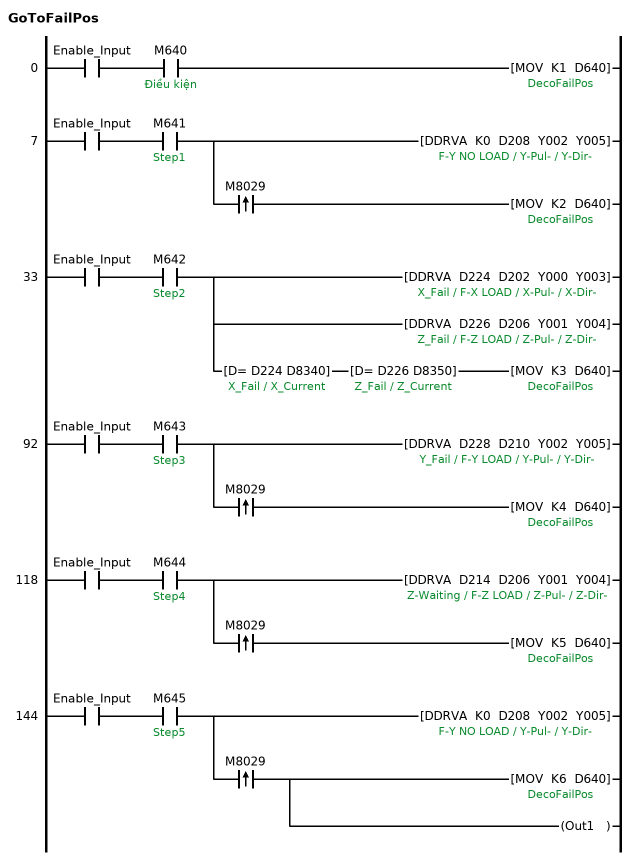
[picture p24: ladder of GoToFailPos, rungs at steps 0 to 144]
0     LD      Enable_Input
      AND     M640  ; Điều kiện
      MOV     K1 D640  ; DecoFailPos
7     LD      Enable_Input
      AND     M641  ; Step1
      DDRVA   K0 D208 Y002 Y005  ; F-Y NO LOAD / Y-Pul- / Y-Dir-
      ANDP    M8029
      MOV     K2 D640
33    LD      Enable_Input
      AND     M642  ; Step2
      DDRVA   D224 D202 Y000 Y003  ; X_Fail / F-X LOAD / X-Pul- / X-Dir-
      DDRVA   D226 D206 Y001 Y004  ; Z_Fail / F-Z LOAD / Z-Pul- / Z-Dir-
      ANDD=   D224 D8340  ; X_Fail / X_Current
      ANDD=   D226 D8350  ; Z_Fail / Z_Current
      MOV     K3 D640
92    LD      Enable_Input
      AND     M643  ; Step3
      DDRVA   D228 D210 Y002 Y005  ; Y_Fail / F-Y LOAD
      ANDP    M8029
      MOV     K4 D640
118   LD      Enable_Input
      AND     M644  ; Step4
      DDRVA   D214 D206 Y001 Y004  ; Z-Waiting
      ANDP    M8029
      MOV     K5 D640
144   LD      Enable_Input
      AND     M645  ; Step5
      DDRVA   K0 D208 Y002 Y005
      ANDP    M8029
      MOV     K6 D640
      OUT     Out1
END_FUNCTION_BLOCK

PROGRAM RETRI
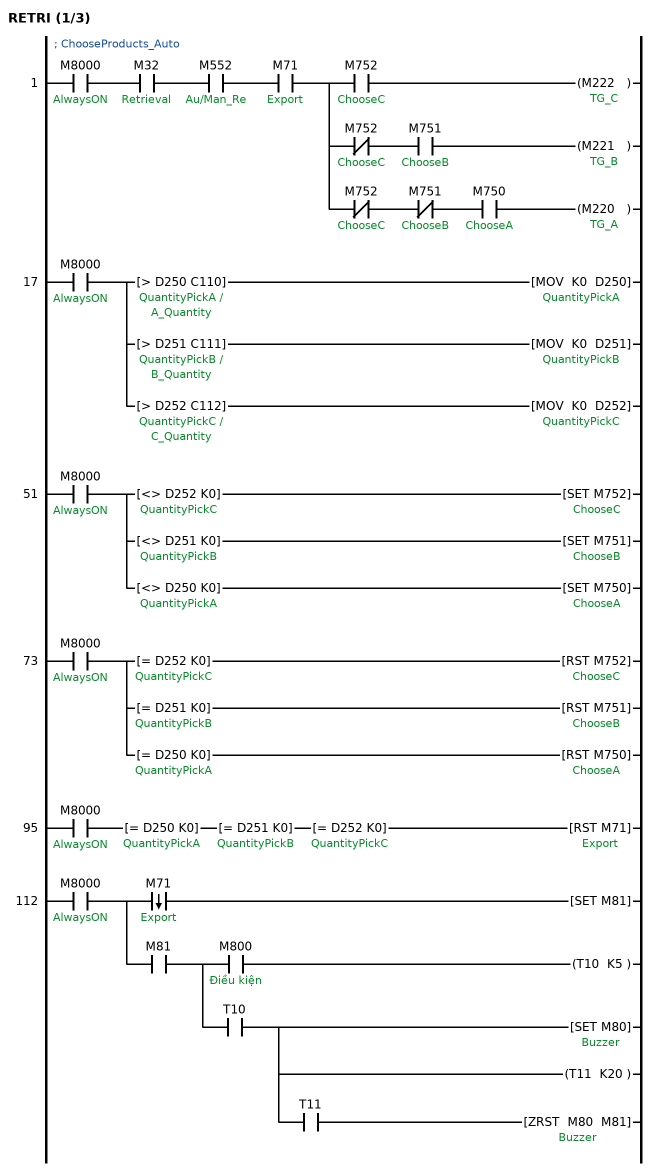
; ChooseProducts_Auto
1     LD      M8000  ; AlwaysON
      AND     M32  ; Retrieval
      AND     M552  ; Au/Man_Re
      AND     M71  ; Export
      MPS
      AND     M752  ; ChooseC
      OUT     M222  ; TG_C
      MRD
      ANI     M752  ; ChooseC
      AND     M751  ; ChooseB
      OUT     M221  ; TG_B
      MPP
      ANI     M752  ; ChooseC
      ANI     M751  ; ChooseB
      AND     M750  ; ChooseA
      OUT     M220  ; TG_A
17    LD      M8000  ; AlwaysON
      MPS
      AND>    D250 C110  ; QuantityPickA / A_Quantity
      MOV     K0 D250
      MRD
      AND>    D251 C111  ; QuantityPickB / B_Quantity
      MOV     K0 D251
      MPP
      AND>    D252 C112  ; QuantityPickC / C_Quantity
      MOV     K0 D252
51    LD      M8000  ; AlwaysON
      MPS
      AND<>   D252 K0  ; QuantityPickC
      SET     M752  ; ChooseC
      MRD
      AND<>   D251 K0  ; QuantityPickB
      SET     M751  ; ChooseB
      MPP
      AND<>   D250 K0  ; QuantityPickA
      SET     M750  ; ChooseA
73    LD      M8000  ; AlwaysON
      MPS
      AND=    D252 K0  ; QuantityPickC
      RST     M752  ; ChooseC
      MRD
      AND=    D251 K0  ; QuantityPickB
      RST     M751  ; ChooseB
      MPP
      AND=    D250 K0  ; QuantityPickA
      RST     M750  ; ChooseA
95    LD      M8000  ; AlwaysON
      AND=    D250 K0  ; QuantityPickA
      AND=    D251 K0  ; QuantityPickB
      AND=    D252 K0  ; QuantityPickC
      RST     M71  ; Export
112   LD      M8000  ; AlwaysON
      MPS
      ANDF    M71  ; Export
      SET     M81
      MPP
      AND     M81
      MPS
      AND     M800  ; Điều kiện
      OUT     T10 K5
      MPP
      AND     T10
      SET     M80  ; Buzzer
      OUT     T11 K20
      AND     T11
      ZRST    M80 M81
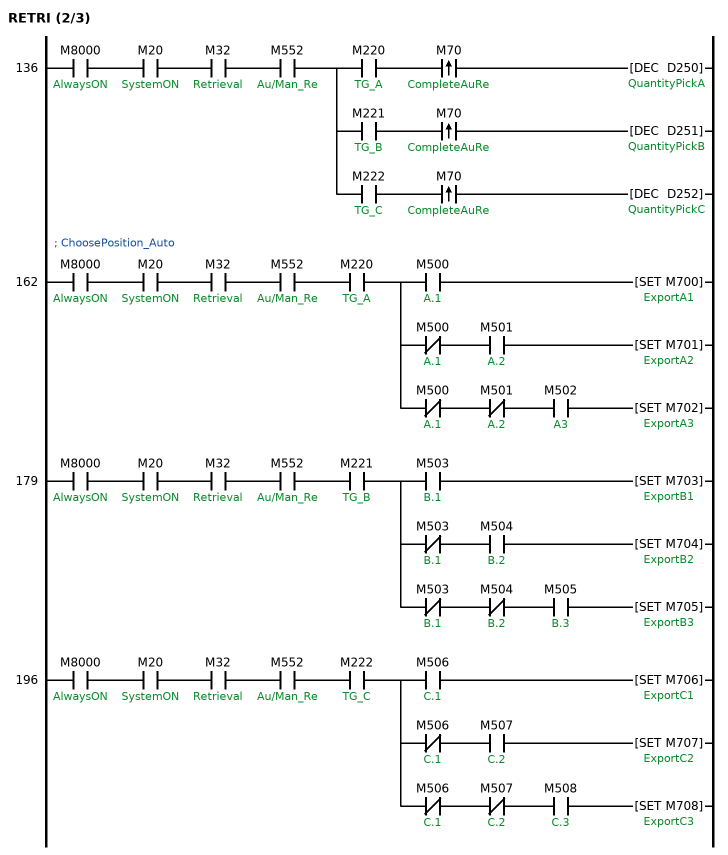
136   LD      M8000  ; AlwaysON
      AND     M20  ; SystemON
      AND     M32  ; Retrieval
      AND     M552  ; Au/Man_Re
      MPS
      AND     M220  ; TG_A
      ANDP    M70  ; CompleteAuRe
      DEC     D250
      MRD
      AND     M221  ; TG_B
      ANDP    M70  ; CompleteAuRe
      DEC     D251
      MPP
      AND     M222  ; TG_C
      ANDP    M70  ; CompleteAuRe
      DEC     D252
; ChoosePosition_Auto
162   LD      M8000  ; AlwaysON
      AND     M20  ; SystemON
      AND     M32  ; Retrieval
      AND     M552  ; Au/Man_Re
      AND     M220  ; TG_A
      MPS
      AND     M500  ; A.1
      SET     M700  ; ExportA1
      MRD
      ANI     M500  ; A.1
      AND     M501  ; A.2
      SET     M701  ; ExportA2
      MPP
      ANI     M500  ; A.1
      ANI     M501  ; A.2
      AND     M502  ; A3
      SET     M702  ; ExportA3
179   LD      M8000  ; AlwaysON
      AND     M20  ; SystemON
      AND     M32  ; Retrieval
      AND     M552  ; Au/Man_Re
      AND     M221  ; TG_B
      MPS
      AND     M503  ; B.1
      SET     M703  ; ExportB1
      MRD
      ANI     M503  ; B.1
      AND     M504  ; B.2
      SET     M704  ; ExportB2
      MPP
      ANI     M503  ; B.1
      ANI     M504  ; B.2
      AND     M505  ; B.3
      SET     M705  ; ExportB3
196   LD      M8000  ; AlwaysON
      AND     M20  ; SystemON
      AND     M32  ; Retrieval
      AND     M552  ; Au/Man_Re
      AND     M222  ; TG_C
      MPS
      AND     M506  ; C.1
      SET     M706  ; ExportC1
      MRD
      ANI     M506  ; C.1
      AND     M507  ; C.2
      SET     M707  ; ExportC2
      MPP
      ANI     M506  ; C.1
      ANI     M507  ; C.2
      AND     M508  ; C.3
      SET     M708  ; ExportC3
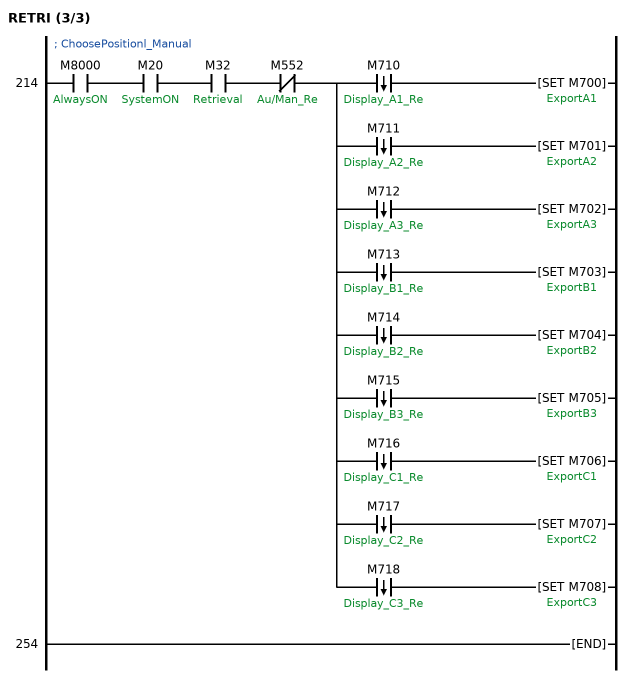
; ChoosePositionl_Manual
214   LD      M8000  ; AlwaysON
      AND     M20  ; SystemON
      AND     M32  ; Retrieval
      ANI     M552  ; Au/Man_Re
      MPS
      ANDF    M710  ; Display_A1_Re
      SET     M700  ; ExportA1
      MRD
      ANDF    M711  ; Display_A2_Re
      SET     M701  ; ExportA2
      MRD
      ANDF    M712  ; Display_A3_Re
      SET     M702  ; ExportA3
      MRD
      ANDF    M713  ; Display_B1_Re
      SET     M703  ; ExportB1
      MRD
      ANDF    M714  ; Display_B2_Re
      SET     M704  ; ExportB2
      MRD
      ANDF    M715  ; Display_B3_Re
      SET     M705  ; ExportB3
      MRD
      ANDF    M716  ; Display_C1_Re
      SET     M706  ; ExportC1
      MRD
      ANDF    M717  ; Display_C2_Re
      SET     M707  ; ExportC2
      MPP
      ANDF    M718  ; Display_C3_Re
      SET     M708  ; ExportC3
254   END
END_PROGRAM

PROGRAM Display
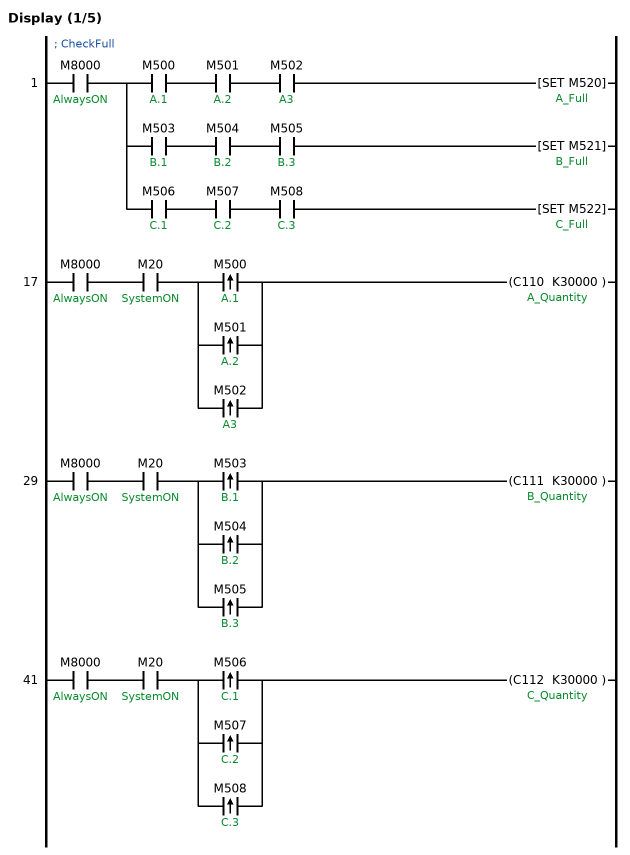
; CheckFull
1     LD      M8000  ; AlwaysON
      MPS
      AND     M500  ; A.1
      AND     M501  ; A.2
      AND     M502  ; A3
      SET     M520  ; A_Full
      MRD
      AND     M503  ; B.1
      AND     M504  ; B.2
      AND     M505  ; B.3
      SET     M521  ; B_Full
      MPP
      AND     M506  ; C.1
      AND     M507  ; C.2
      AND     M508  ; C.3
      SET     M522  ; C_Full
17    LD      M8000  ; AlwaysON
      AND     M20  ; SystemON
      LDP     M500  ; A.1
      ORP     M501  ; A.2
      ORP     M502  ; A3
      ANB
      OUT     C110 K30000  ; A_Quantity
29    LD      M8000  ; AlwaysON
      AND     M20  ; SystemON
      LDP     M503  ; B.1
      ORP     M504  ; B.2
      ORP     M505  ; B.3
      ANB
      OUT     C111 K30000  ; B_Quantity
41    LD      M8000  ; AlwaysON
      AND     M20  ; SystemON
      LDP     M506  ; C.1
      ORP     M507  ; C.2
      ORP     M508  ; C.3
      ANB
      OUT     C112 K30000  ; C_Quantity
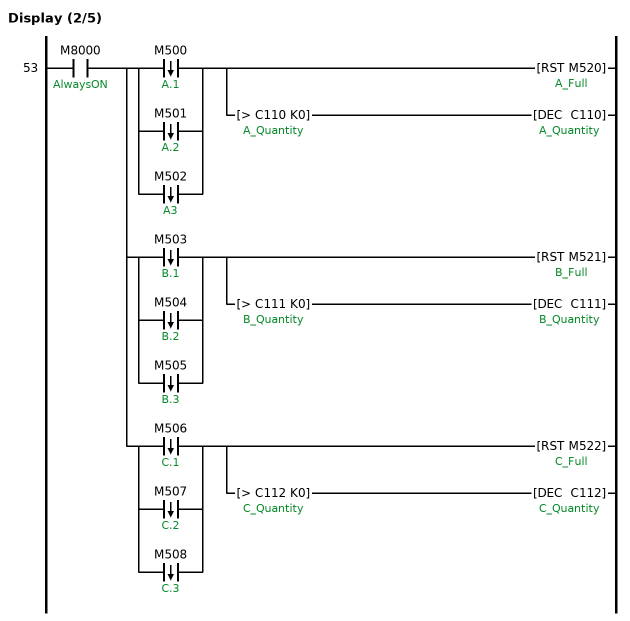
53    LD      M8000  ; AlwaysON
      MPS
      LDF     M500  ; A.1
      ORF     M501  ; A.2
      ORF     M502  ; A3
      ANB
      RST     M520  ; A_Full
      AND>    C110 K0  ; A_Quantity
      DEC     C110
      MRD
      LDF     M503  ; B.1
      ORF     M504  ; B.2
      ORF     M505  ; B.3
      ANB
      RST     M521  ; B_Full
      AND>    C111 K0  ; B_Quantity
      DEC     C111
      MPP
      LDF     M506  ; C.1
      ORF     M507  ; C.2
      ORF     M508  ; C.3
      ANB
      RST     M522  ; C_Full
      AND>    C112 K0  ; C_Quantity
      DEC     C112
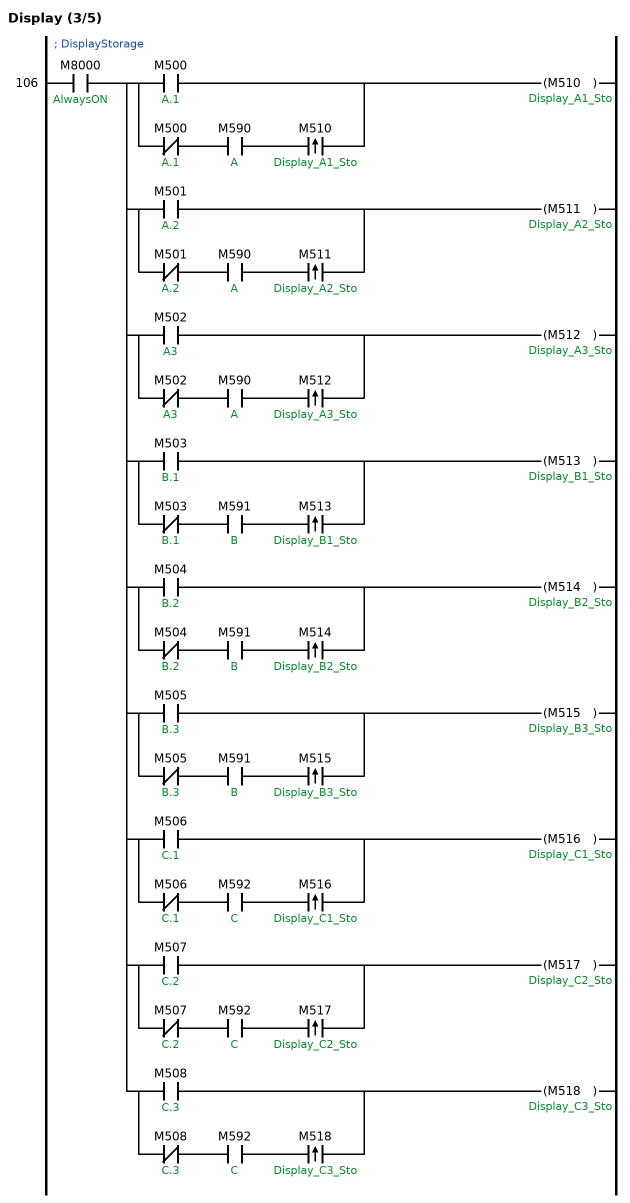
; DisplayStorage
106   LD      M8000  ; AlwaysON
      MPS
      LD      M500  ; A.1
      LDI     M500  ; A.1
      AND     M590  ; A
      ANDP    M510  ; Display_A1_Sto
      ORB
      ANB
      OUT     M510  ; Display_A1_Sto
      MRD
      LD      M501  ; A.2
      LDI     M501  ; A.2
      AND     M590  ; A
      ANDP    M511  ; Display_A2_Sto
      ORB
      ANB
      OUT     M511  ; Display_A2_Sto
      MRD
      LD      M502  ; A3
      LDI     M502  ; A3
      AND     M590  ; A
      ANDP    M512  ; Display_A3_Sto
      ORB
      ANB
      OUT     M512  ; Display_A3_Sto
      MRD
      LD      M503  ; B.1
      LDI     M503  ; B.1
      AND     M591  ; B
      ANDP    M513  ; Display_B1_Sto
      ORB
      ANB
      OUT     M513  ; Display_B1_Sto
      MRD
      LD      M504  ; B.2
      LDI     M504  ; B.2
      AND     M591  ; B
      ANDP    M514  ; Display_B2_Sto
      ORB
      ANB
      OUT     M514  ; Display_B2_Sto
      MRD
      LD      M505  ; B.3
      LDI     M505  ; B.3
      AND     M591  ; B
      ANDP    M515  ; Display_B3_Sto
      ORB
      ANB
      OUT     M515  ; Display_B3_Sto
      MRD
      LD      M506  ; C.1
      LDI     M506  ; C.1
      AND     M592  ; C
      ANDP    M516  ; Display_C1_Sto
      ORB
      ANB
      OUT     M516  ; Display_C1_Sto
      MRD
      LD      M507  ; C.2
      LDI     M507  ; C.2
      AND     M592  ; C
      ANDP    M517  ; Display_C2_Sto
      ORB
      ANB
      OUT     M517  ; Display_C2_Sto
      MPP
      LD      M508  ; C.3
      LDI     M508  ; C.3
      AND     M592  ; C
      ANDP    M518  ; Display_C3_Sto
      ORB
      ANB
      OUT     M518  ; Display_C3_Sto
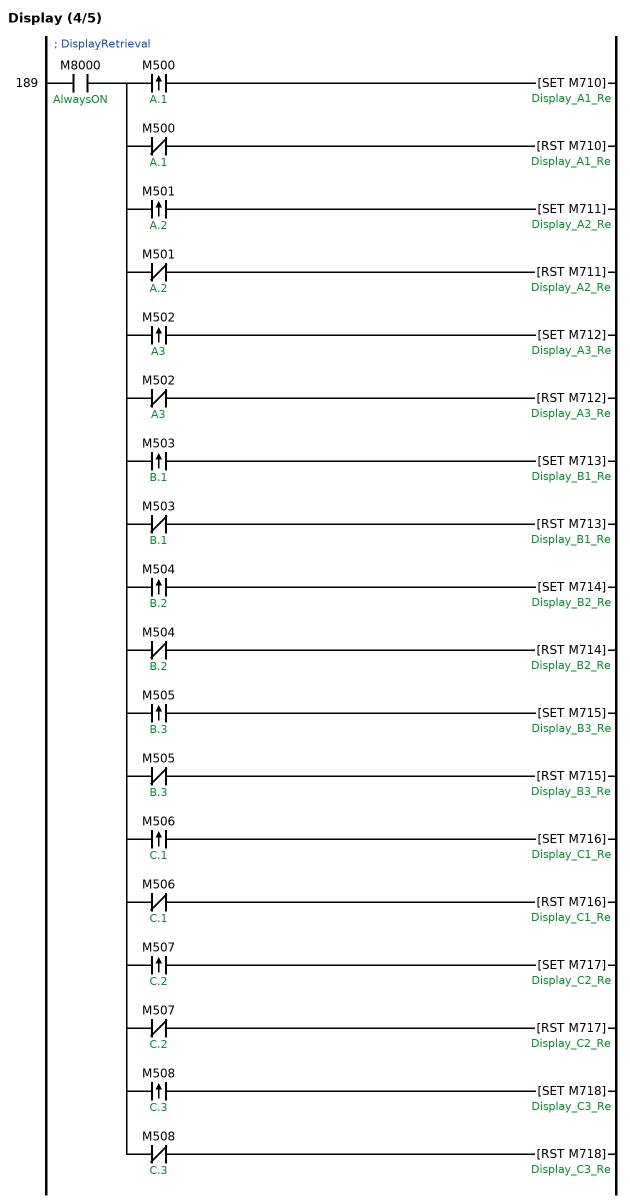
; DisplayRetrieval
189   LD      M8000  ; AlwaysON
      MPS
      ANDP    M500  ; A.1
      SET     M710  ; Display_A1_Re
      MRD
      ANI     M500  ; A.1
      RST     M710  ; Display_A1_Re
      MRD
      ANDP    M501  ; A.2
      SET     M711  ; Display_A2_Re
      MRD
      ANI     M501  ; A.2
      RST     M711  ; Display_A2_Re
      MRD
      ANDP    M502  ; A3
      SET     M712  ; Display_A3_Re
      MRD
      ANI     M502  ; A3
      RST     M712  ; Display_A3_Re
      MRD
      ANDP    M503  ; B.1
      SET     M713  ; Display_B1_Re
      MRD
      ANI     M503  ; B.1
      RST     M713  ; Display_B1_Re
      MRD
      ANDP    M504  ; B.2
      SET     M714  ; Display_B2_Re
      MRD
      ANI     M504  ; B.2
      RST     M714  ; Display_B2_Re
      MRD
      ANDP    M505  ; B.3
      SET     M715  ; Display_B3_Re
      MRD
      ANI     M505  ; B.3
      RST     M715  ; Display_B3_Re
      MRD
      ANDP    M506  ; C.1
      SET     M716  ; Display_C1_Re
      MRD
      ANI     M506  ; C.1
      RST     M716  ; Display_C1_Re
      MRD
      ANDP    M507  ; C.2
      SET     M717  ; Display_C2_Re
      MRD
      ANI     M507  ; C.2
      RST     M717  ; Display_C2_Re
      MRD
      ANDP    M508  ; C.3
      SET     M718  ; Display_C3_Re
      MPP
      ANI     M508  ; C.3
      RST     M718  ; Display_C3_Re
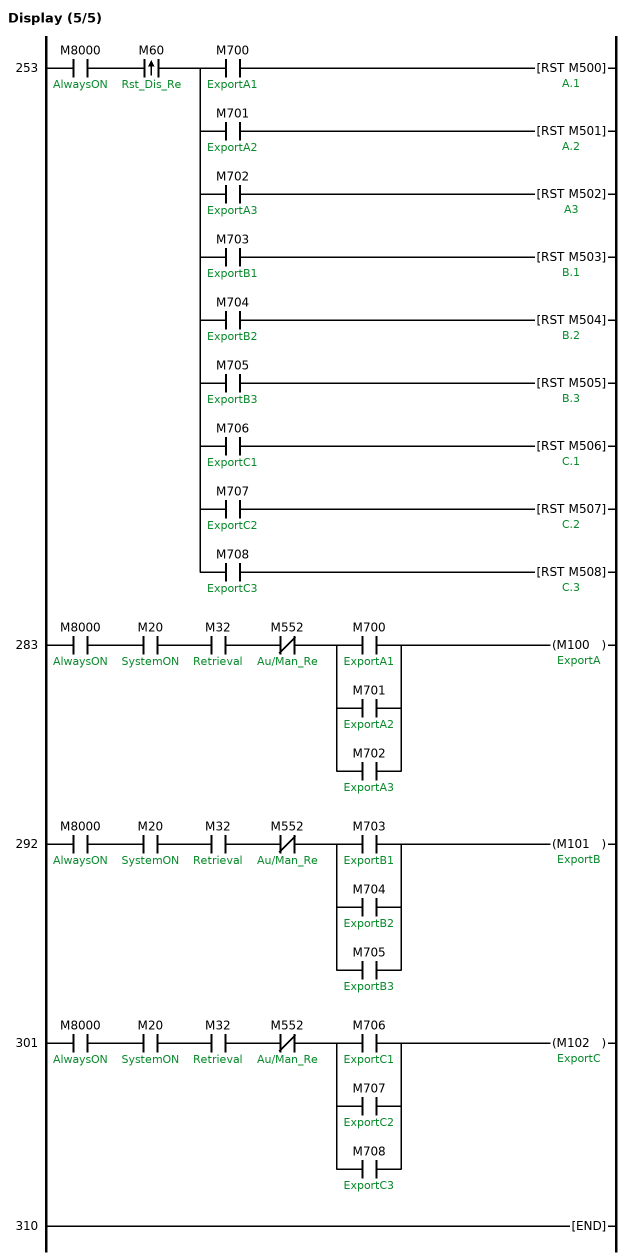
253   LD      M8000  ; AlwaysON
      ANDP    M60  ; Rst_Dis_Re
      MPS
      AND     M700  ; ExportA1
      RST     M500  ; A.1
      MRD
      AND     M701  ; ExportA2
      RST     M501  ; A.2
      MRD
      AND     M702  ; ExportA3
      RST     M502  ; A3
      MRD
      AND     M703  ; ExportB1
      RST     M503  ; B.1
      MRD
      AND     M704  ; ExportB2
      RST     M504  ; B.2
      MRD
      AND     M705  ; ExportB3
      RST     M505  ; B.3
      MRD
      AND     M706  ; ExportC1
      RST     M506  ; C.1
      MRD
      AND     M707  ; ExportC2
      RST     M507  ; C.2
      MPP
      AND     M708  ; ExportC3
      RST     M508  ; C.3
283   LD      M8000  ; AlwaysON
      AND     M20  ; SystemON
      AND     M32  ; Retrieval
      ANI     M552  ; Au/Man_Re
      LD      M700  ; ExportA1
      OR      M701  ; ExportA2
      OR      M702  ; ExportA3
      ANB
      OUT     M100  ; ExportA
292   LD      M8000  ; AlwaysON
      AND     M20  ; SystemON
      AND     M32  ; Retrieval
      ANI     M552  ; Au/Man_Re
      LD      M703  ; ExportB1
      OR      M704  ; ExportB2
      OR      M705  ; ExportB3
      ANB
      OUT     M101  ; ExportB
301   LD      M8000  ; AlwaysON
      AND     M20  ; SystemON
      AND     M32  ; Retrieval
      ANI     M552  ; Au/Man_Re
      LD      M706  ; ExportC1
      OR      M707  ; ExportC2
      OR      M708  ; ExportC3
      ANB
      OUT     M102  ; ExportC
310   END
END_PROGRAM

PROGRAM STO
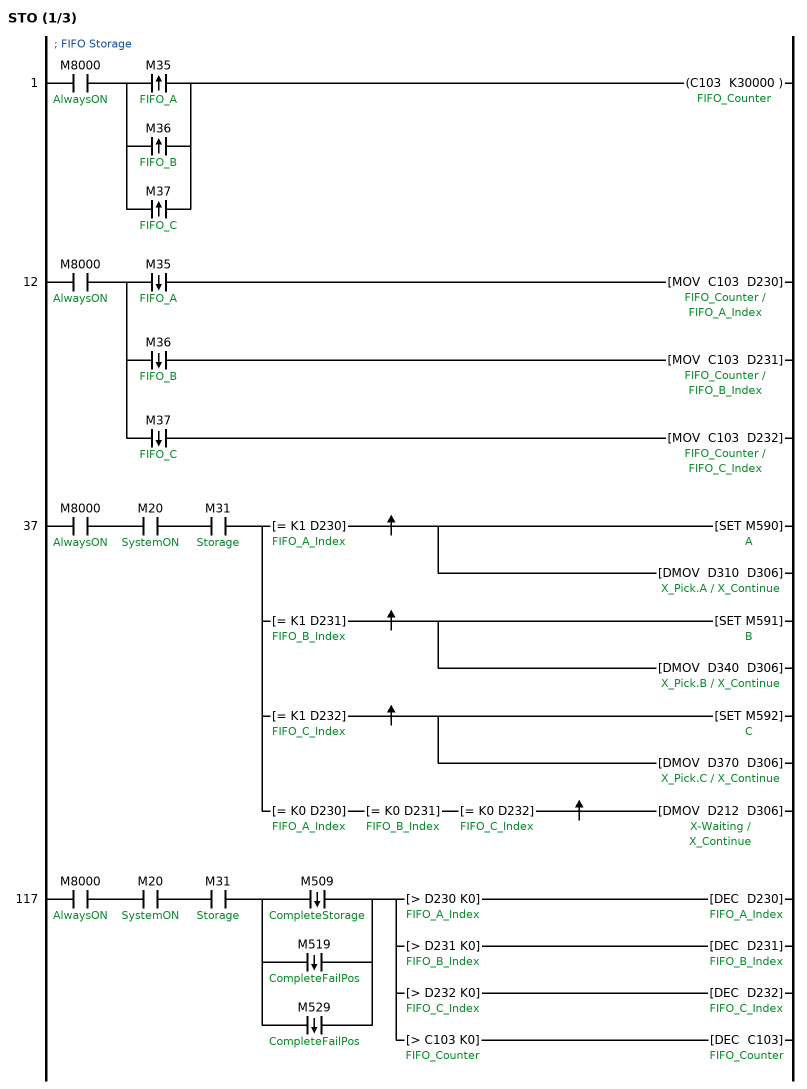
; FIFO Storage
1     LD      M8000  ; AlwaysON
      LDP     M35  ; FIFO_A
      ORP     M36  ; FIFO_B
      ORP     M37  ; FIFO_C
      ANB
      OUT     C103 K30000  ; FIFO_Counter
12    LD      M8000  ; AlwaysON
      MPS
      ANDF    M35  ; FIFO_A
      MOV     C103 D230  ; FIFO_A_Index
      MRD
      ANDF    M36  ; FIFO_B
      MOV     C103 D231  ; FIFO_B_Index
      MPP
      ANDF    M37  ; FIFO_C
      MOV     C103 D232  ; FIFO_C_Index
37    LD      M8000  ; AlwaysON
      AND     M20  ; SystemON
      AND     M31  ; Storage
      MPS
      AND=    K1 D230  ; FIFO_A_Index
      MEP
      SET     M590  ; A
      DMOV    D310 D306  ; X_Pick.A / X_Continue
      MRD
      AND=    K1 D231  ; FIFO_B_Index
      MEP
      SET     M591  ; B
      DMOV    D340 D306  ; X_Pick.B
      MRD
      AND=    K1 D232  ; FIFO_C_Index
      MEP
      SET     M592  ; C
      DMOV    D370 D306  ; X_Pick.C
      MPP
      AND=    K0 D230  ; FIFO_A_Index
      AND=    K0 D231  ; FIFO_B_Index
      AND=    K0 D232  ; FIFO_C_Index
      MEP
      DMOV    D212 D306  ; X-Waiting
117   LD      M8000  ; AlwaysON
      AND     M20  ; SystemON
      AND     M31  ; Storage
      LDF     M509  ; CompleteStorage
      ORF     M519  ; CompleteFailPos
      ORF     M529  ; CompleteFailPos
      ANB
      MPS
      AND>    D230 K0  ; FIFO_A_Index
      DEC     D230
      MRD
      AND>    D231 K0  ; FIFO_B_Index
      DEC     D231
      MRD
      AND>    D232 K0  ; FIFO_C_Index
      DEC     D232
      MPP
      AND>    C103 K0  ; FIFO_Counter
      DEC     C103
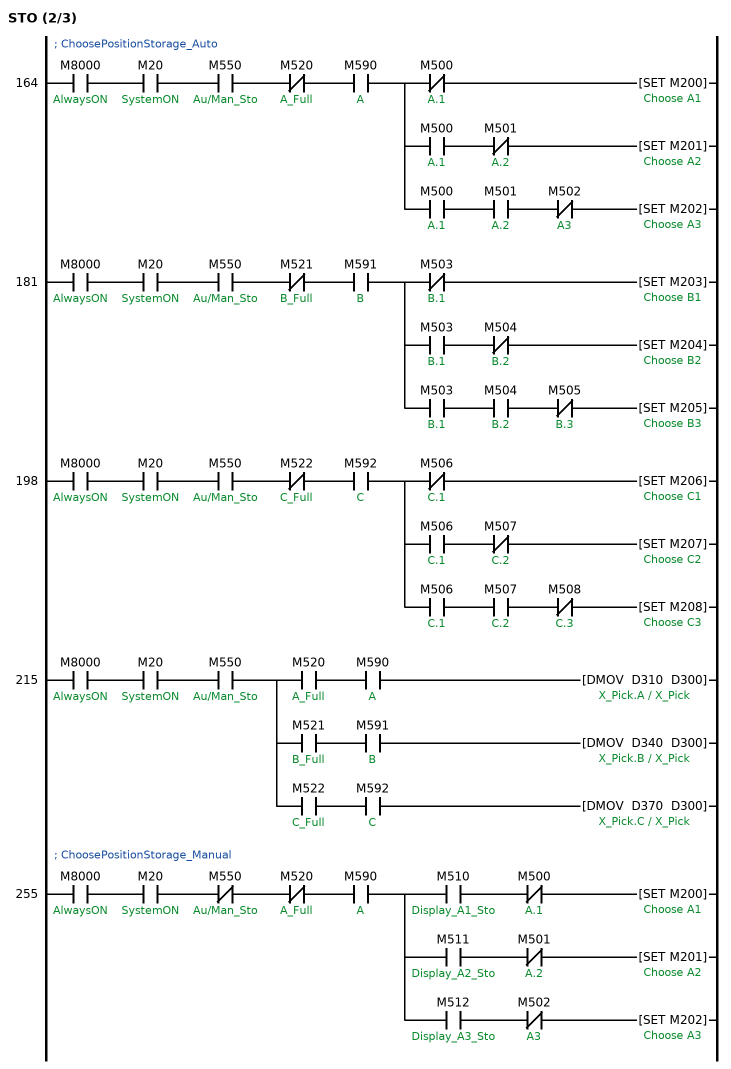
; ChoosePositionStorage_Auto
164   LD      M8000  ; AlwaysON
      AND     M20  ; SystemON
      AND     M550  ; Au/Man_Sto
      ANI     M520  ; A_Full
      AND     M590  ; A
      MPS
      ANI     M500  ; A.1
      SET     M200  ; Choose A1
      MRD
      AND     M500  ; A.1
      ANI     M501  ; A.2
      SET     M201  ; Choose A2
      MPP
      AND     M500  ; A.1
      AND     M501  ; A.2
      ANI     M502  ; A3
      SET     M202  ; Choose A3
181   LD      M8000  ; AlwaysON
      AND     M20  ; SystemON
      AND     M550  ; Au/Man_Sto
      ANI     M521  ; B_Full
      AND     M591  ; B
      MPS
      ANI     M503  ; B.1
      SET     M203  ; Choose B1
      MRD
      AND     M503  ; B.1
      ANI     M504  ; B.2
      SET     M204  ; Choose B2
      MPP
      AND     M503  ; B.1
      AND     M504  ; B.2
      ANI     M505  ; B.3
      SET     M205  ; Choose B3
198   LD      M8000  ; AlwaysON
      AND     M20  ; SystemON
      AND     M550  ; Au/Man_Sto
      ANI     M522  ; C_Full
      AND     M592  ; C
      MPS
      ANI     M506  ; C.1
      SET     M206  ; Choose C1
      MRD
      AND     M506  ; C.1
      ANI     M507  ; C.2
      SET     M207  ; Choose C2
      MPP
      AND     M506  ; C.1
      AND     M507  ; C.2
      ANI     M508  ; C.3
      SET     M208  ; Choose C3
215   LD      M8000  ; AlwaysON
      AND     M20  ; SystemON
      AND     M550  ; Au/Man_Sto
      MPS
      AND     M520  ; A_Full
      AND     M590  ; A
      DMOV    D310 D300  ; X_Pick
      MRD
      AND     M521  ; B_Full
      AND     M591  ; B
      DMOV    D340 D300
      MPP
      AND     M522  ; C_Full
      AND     M592  ; C
      DMOV    D370 D300
; ChoosePositionStorage_Manual
255   LD      M8000  ; AlwaysON
      AND     M20  ; SystemON
      ANI     M550  ; Au/Man_Sto
      ANI     M520  ; A_Full
      AND     M590  ; A
      MPS
      AND     M510  ; Display_A1_Sto
      ANI     M500  ; A.1
      SET     M200  ; Choose A1
      MRD
      AND     M511  ; Display_A2_Sto
      ANI     M501  ; A.2
      SET     M201  ; Choose A2
      MPP
      AND     M512  ; Display_A3_Sto
      ANI     M502  ; A3
      SET     M202  ; Choose A3
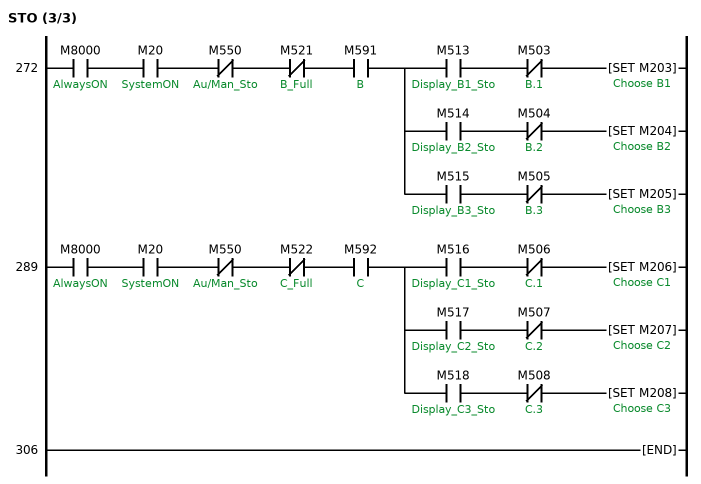
272   LD      M8000  ; AlwaysON
      AND     M20  ; SystemON
      ANI     M550  ; Au/Man_Sto
      ANI     M521  ; B_Full
      AND     M591  ; B
      MPS
      AND     M513  ; Display_B1_Sto
      ANI     M503  ; B.1
      SET     M203  ; Choose B1
      MRD
      AND     M514  ; Display_B2_Sto
      ANI     M504  ; B.2
      SET     M204  ; Choose B2
      MPP
      AND     M515  ; Display_B3_Sto
      ANI     M505  ; B.3
      SET     M205  ; Choose B3
289   LD      M8000  ; AlwaysON
      AND     M20  ; SystemON
      ANI     M550  ; Au/Man_Sto
      ANI     M522  ; C_Full
      AND     M592  ; C
      MPS
      AND     M516  ; Display_C1_Sto
      ANI     M506  ; C.1
      SET     M206  ; Choose C1
      MRD
      AND     M517  ; Display_C2_Sto
      ANI     M507  ; C.2
      SET     M207  ; Choose C2
      MPP
      AND     M518  ; Display_C3_Sto
      ANI     M508  ; C.3
      SET     M208  ; Choose C3
306   END
END_PROGRAM

// device comments not shown above
X004  ; X++
X006  ; Z++
X010  ; Y++
M33  ; Fault
M530  ; A_FIFO
M531  ; B_FIFO
M532  ; C_FIFO
M540  ; InvertA
M541  ; InvertB
M542  ; InvertC
M647  ; Step7
M648  ; Step8
M649  ; Step9
M709  ; CompleteRetrieval
M760  ; tgA
M761  ; tgB
M762  ; tgB
M811  ; Step11
D0  ; Screen
D234  ; Y_Waiting
D350  ; X_Pick.B2
D408  ; Y_Place
